FUNCTION_BLOCK FINAL FB
VAR_INPUT
END_VAR
VAR_OUTPUT
END_VAR
VAR
END_VAR

END_FUNCTION_BLOCK

(* stored: Version 1.1.0.1, ProductVersion 3.1.4024.12
   POU FB: Id {570d6aa9-2f59-4dc1-8b37-85e86c9336c8}, SpecialFunc None *)
